FUNCTION_BLOCK CrossJoystick (* Basic FB representing a Cross-Joystick *)
  (* Standard: 61499-2 *)
  (* Version 1.0, 2026-06-15, Antigravity, 4DIAC-Consortium *)
  PACKAGE logiBUS::utils::sequence::joystick;
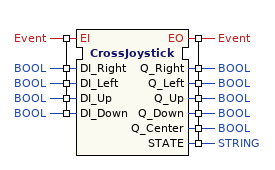
  EVENT_INPUT
    EI WITH DI_Right, DI_Left, DI_Up, DI_Down; (* Event input for state changes *)
  END_EVENT
  EVENT_OUTPUT
    EO WITH Q_Right, Q_Left, Q_Up, Q_Down, Q_Center, STATE; (* Event output indicating state execution *)
  END_EVENT
  VAR_INPUT
    DI_Right : BOOL; (* Joystick moved Right *)
    DI_Left : BOOL; (* Joystick moved Left *)
    DI_Up : BOOL; (* Joystick moved Up *)
    DI_Down : BOOL; (* Joystick moved Down *)
  END_VAR
  VAR_OUTPUT
    Q_Right : BOOL; (* Output indicating Right state *)
    Q_Left : BOOL; (* Output indicating Left state *)
    Q_Up : BOOL; (* Output indicating Up state *)
    Q_Down : BOOL; (* Output indicating Down state *)
    Q_Center : BOOL; (* Output indicating Center state *)
    STATE : STRING; (* Current state name *)
  END_VAR
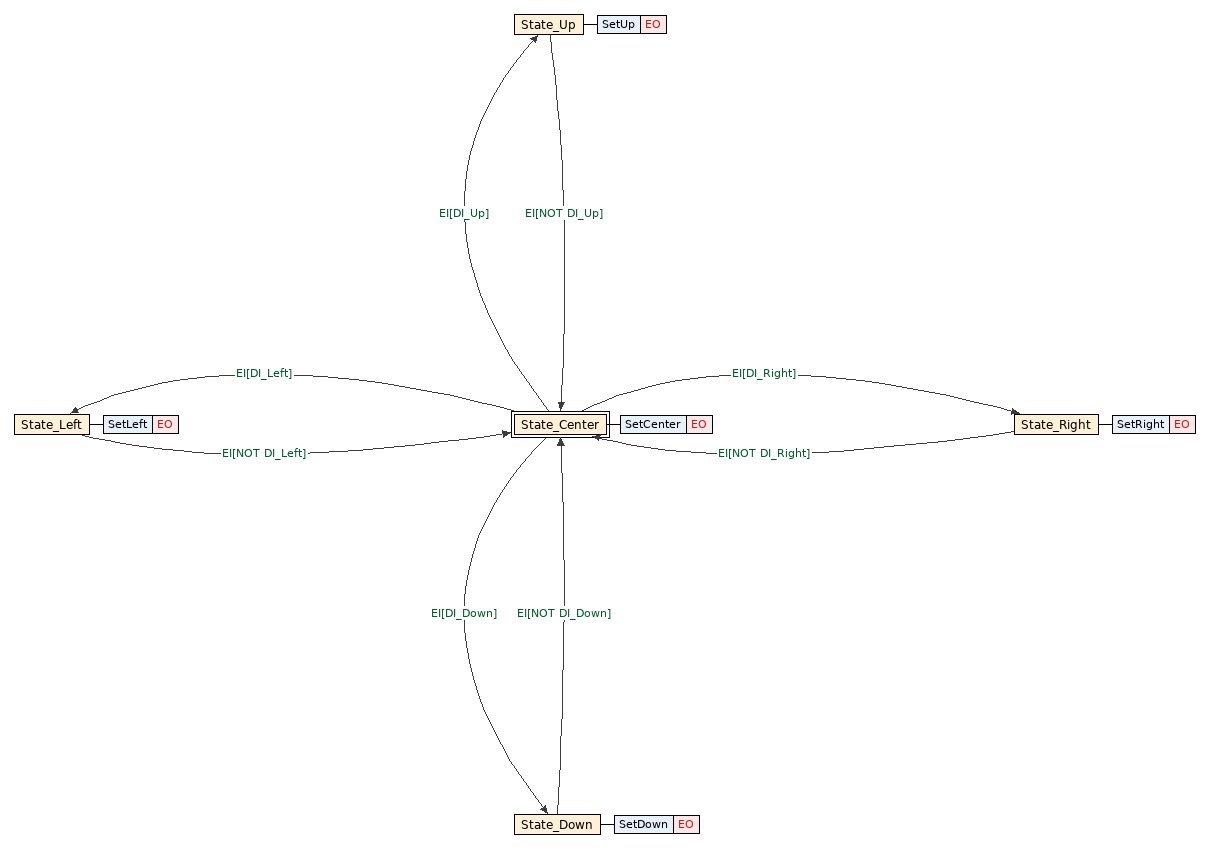
  EC_STATES
    State_Center : SetCenter -> EO; (* Initial State (Joystick in center) *)
    State_Right : SetRight -> EO; (* Joystick in Right state *)
    State_Left : SetLeft -> EO; (* Joystick in Left state *)
    State_Up : SetUp -> EO; (* Joystick in Up state *)
    State_Down : SetDown -> EO; (* Joystick in Down state *)
  END_STATES
  EC_TRANSITIONS
    State_Center TO State_Right := EI[DI_Right]; (* Move Right *)
    State_Center TO State_Left := EI[DI_Left]; (* Move Left *)
    State_Center TO State_Up := EI[DI_Up]; (* Move Up *)
    State_Center TO State_Down := EI[DI_Down]; (* Move Down *)
    State_Right TO State_Center := EI[NOT DI_Right]; (* Return to Center *)
    State_Left TO State_Center := EI[NOT DI_Left]; (* Return to Center *)
    State_Up TO State_Center := EI[NOT DI_Up]; (* Return to Center *)
    State_Down TO State_Center := EI[NOT DI_Down]; (* Return to Center *)
  END_TRANSITIONS
  ALGORITHM SetCenter IN ST: (* Set Center Outputs *)
Q_Right := BOOL#FALSE;
Q_Left := BOOL#FALSE;
Q_Up := BOOL#FALSE;
Q_Down := BOOL#FALSE;
Q_Center := BOOL#TRUE;
STATE := 'Center';
  END_ALGORITHM
  ALGORITHM SetRight IN ST: (* Set Right Outputs *)
Q_Right := BOOL#TRUE;
Q_Left := BOOL#FALSE;
Q_Up := BOOL#FALSE;
Q_Down := BOOL#FALSE;
Q_Center := BOOL#FALSE;
STATE := 'Right';
  END_ALGORITHM
  ALGORITHM SetLeft IN ST: (* Set Left Outputs *)
Q_Right := BOOL#FALSE;
Q_Left := BOOL#TRUE;
Q_Up := BOOL#FALSE;
Q_Down := BOOL#FALSE;
Q_Center := BOOL#FALSE;
STATE := 'Left';
  END_ALGORITHM
  ALGORITHM SetUp IN ST: (* Set Up Outputs *)
Q_Right := BOOL#FALSE;
Q_Left := BOOL#FALSE;
Q_Up := BOOL#TRUE;
Q_Down := BOOL#FALSE;
Q_Center := BOOL#FALSE;
STATE := 'Up';
  END_ALGORITHM
  ALGORITHM SetDown IN ST: (* Set Down Outputs *)
Q_Right := BOOL#FALSE;
Q_Left := BOOL#FALSE;
Q_Up := BOOL#FALSE;
Q_Down := BOOL#TRUE;
Q_Center := BOOL#FALSE;
STATE := 'Down';
  END_ALGORITHM
END_FUNCTION_BLOCK
(* other elements stored in the file *)
(* Transitions from Center to directions *)
(* Transitions from directions back to Center (no direct cross transitions allowed) *)
